Fanuc KAREL source: kt00870.KL

-- PROVISIONAL review KL for V770-1; original PC SHA256 5f28812f8aa9d96decb3ce3dc6e1c59a75feb099f0141ea3ca17c45fe48b5094
-- Incomplete behavior may be omitted. Consult companion uncertainty JSON. Do not deploy.
PROGRAM KT00870
%NOLOCKGROUP
VAR
  R1 : REAL
  R2 : REAL
  OUT : INTEGER
BEGIN
  -- UNRESOLVED_PC offsets 5-16; opcodes 2E,23
  -- UNRESOLVED_PC offsets 21-32; opcodes 2E,23
  -- UNRESOLVED_PC offsets 37-48; opcodes 2E,23
  -- UNRESOLVED_PC offsets 53-64; opcodes 2E,23
  -- UNRESOLVED_PC offsets 69-84; opcodes 27,22,76,23
  -- UNRESOLVED_PC offsets 89-93; opcodes 7F
END KT00870
